% RSLogix 500 project I2P JOB 00 - TEMPLATE.RSS, saved by version 10.00.00.00 %
PROJECT "UNTITLED"    % processor: Bul.1763 MicroLogix 1100 Series B %

PROGRAM FILES
  LAD 2 "MAIN"  6 rungs
  LAD 3 "SIM"  12 rungs
  LAD 4 "MTR"  5 rungs  % ESTOP/Stop/Start Motor %
  LAD 5   2 rungs

DATA FILES
  O0 OUTPUT  4 elements
  I1 INPUT  6 elements
  S2 STATUS  66 elements
  B3 BINARY  12 elements
  T4 TIMER  14 elements
  C5 COUNTER  1 elements
  R6 CONTROL  1 elements
  N7 INTEGER  1 elements
  F8 FLOAT  1 elements

LADDER 2 "MAIN"
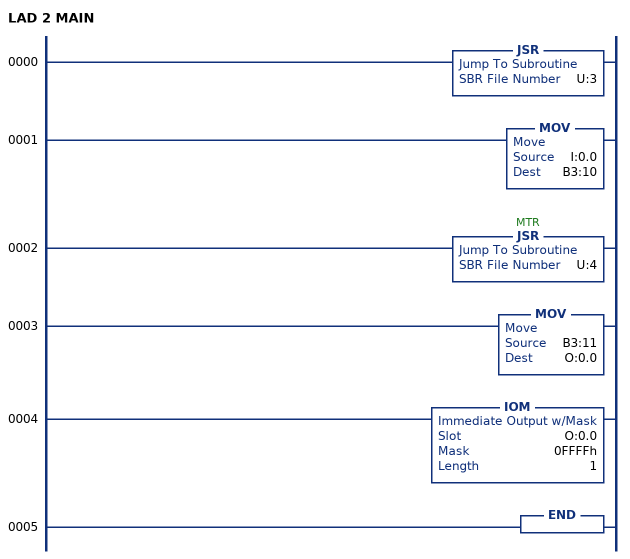
% Rung: 0 %
SOR JSR U:3 EOR
% Rung: 1 %
SOR MOV I:0.0 B3:10 EOR
% Rung: 2 %
SOR JSR U:4 EOR
%   U:4  MTR %
% Rung: 3 %
SOR MOV B3:11 O:0.0 EOR
% Rung: 4 %
SOR IOM O:0.0 0FFFFh 1 EOR
% Rung: 5 %
SOR END EOR

LADDER 3 "SIM"
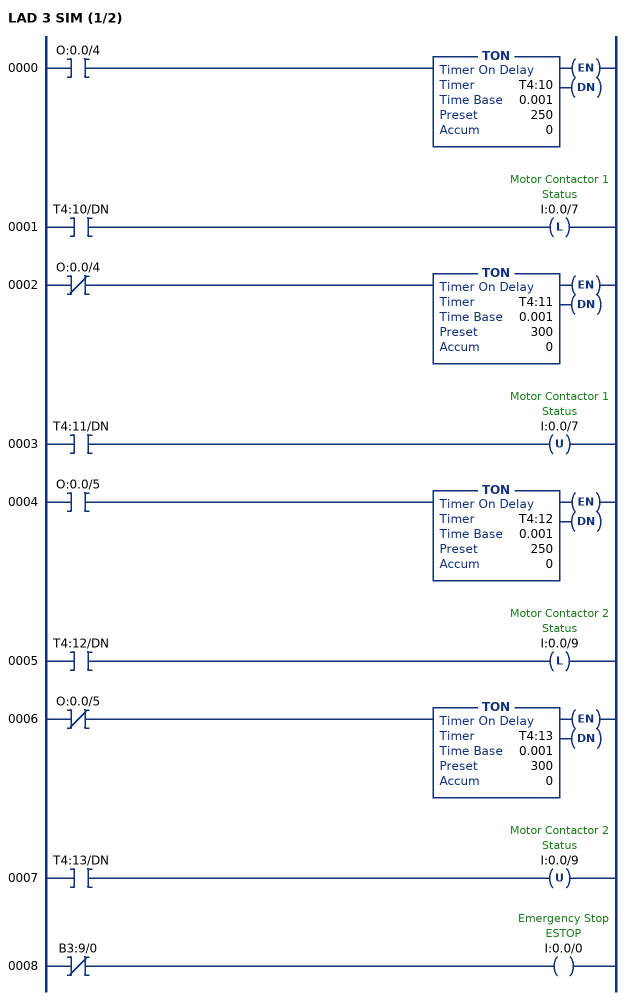
% Rung: 0 %
SOR XIC O:0.0/4 TON T4:10 0.001 250 0 EOR
% Rung: 1 %
SOR XIC T4:10/DN OTL I:0.0/7 EOR
%   I:0.0/7  "Motor Contactor 1 Status" %
% Rung: 2 %
SOR XIO O:0.0/4 TON T4:11 0.001 300 0 EOR
% Rung: 3 %
SOR XIC T4:11/DN OTU I:0.0/7 EOR
%   I:0.0/7  "Motor Contactor 1 Status" %
% Rung: 4 %
SOR XIC O:0.0/5 TON T4:12 0.001 250 0 EOR
% Rung: 5 %
SOR XIC T4:12/DN OTL I:0.0/9 EOR
%   I:0.0/9  "Motor Contactor 2 Status" %
% Rung: 6 %
SOR XIO O:0.0/5 TON T4:13 0.001 300 0 EOR
% Rung: 7 %
SOR XIC T4:13/DN OTU I:0.0/9 EOR
%   I:0.0/9  "Motor Contactor 2 Status" %
% Rung: 8 %
SOR XIO B3:9/0 OTE I:0.0/0 EOR
%   I:0.0/0  ESTOP  "Emergency Stop" %

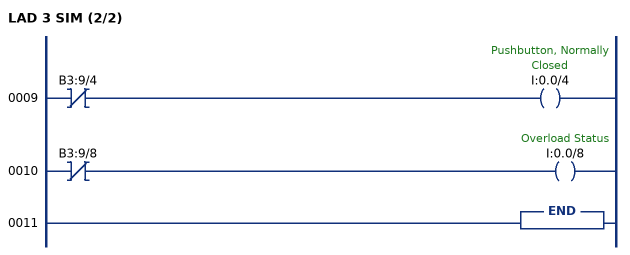
% Rung: 9 %
SOR XIO B3:9/4 OTE I:0.0/4 EOR
%   I:0.0/4  "Pushbutton, Normally Closed" %
% Rung: 10 %
SOR XIO B3:9/8 OTE I:0.0/8 EOR
%   I:0.0/8  "Overload Status" %
% Rung: 11 %
SOR END EOR

LADDER 4 "MTR"    % ESTOP/Stop/Start Motor %
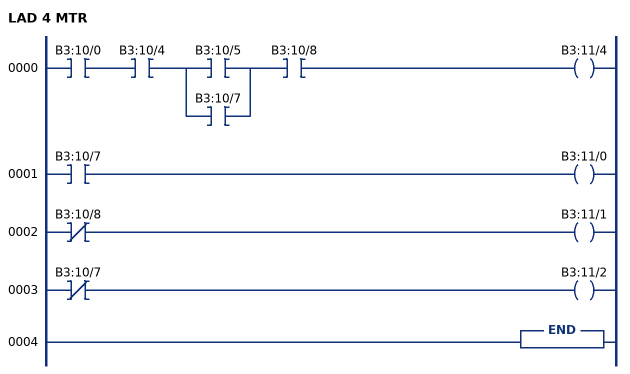
% Rung: 0 %
SOR XIC B3:10/0 XIC B3:10/4 BST XIC B3:10/5 NXB XIC B3:10/7 BND XIC B3:10/8 OTE B3:11/4 EOR
% Rung: 1 %
SOR XIC B3:10/7 OTE B3:11/0 EOR
% Rung: 2 %
SOR XIO B3:10/8 OTE B3:11/1 EOR
% Rung: 3 %
SOR XIO B3:10/7 OTE B3:11/2 EOR
% Rung: 4 %
SOR END EOR

LADDER 5
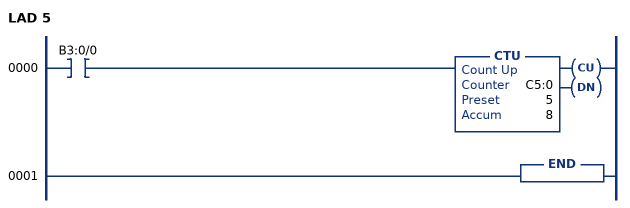
% Rung: 0 %
SOR XIC B3:0/0 CTU C5:0 5 8 EOR
% Rung: 1 %
SOR END EOR

OTHER DOCUMENTED ADDRESSES
  I:0.0/1  "3 Position Selector Switch, Position A"
  I:0.0/2  "3 Position Selector Switch, Position B"
  I:0.0/3  "2 Position Selector Switch, Position A = ON"
  I:0.0/5  "Pushbutton, Normamlly Open"
  I:0.0/6  "Pushbutton, Normamlly Open"
  O:0.0/0  I

DATA TABLE (non-zero values as saved)
DATA B3
% B3:0 % 0X0001 0X0000 0X0000 0X0000 0X0000 0X0000 0X0000 0X0000 0X0000 0X0000
% B3:10 % 0X01A1 0X0000
DATA T4
% .PRE .ACC %
% T4:10 % 250 0
% T4:11 % 300 0
% T4:12 % 250 0
% T4:13 % 300 0
DATA C5
% .PRE .ACC %
% C5:0 % 5 8
